FUNCTION_BLOCK OPCUA_CONNECT_13434D741E95123C0 (* Generic Interface Function Block Type *)
  (* Standard: 61499-2 *)
  (* Version 0.0, 20/09/2020, Administrator, nxtControl GmbH, Template *)
  PACKAGE Main;
  (* Compiler Cpp nxtControl builtin 1.0 *)
  {SET_ATTRIBUTE(Runtime.FBType.ImplementingType, Standard.OPCUAClient#DYNGEN_OPCUA_CONNECT)}
  {SET_ATTRIBUTE(Configuration.GenericFBType.InterfaceParams, Standard.OPCUAClient#CNTX:=1)}
  {SET_ATTRIBUTE(Configuration.FBType.IsKind.OPCUA_CLIENT, )}
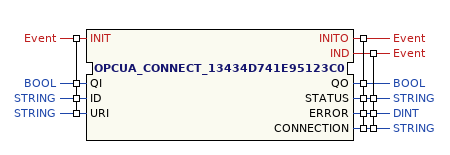
  EVENT_INPUT
    INIT WITH QI, ID, URI; (* Initialization or deinitialization of connection *)
  END_EVENT
  EVENT_OUTPUT
    INITO WITH QO, STATUS, ERROR, CONNECTION; (* Initialization or deinitialization confirmation event *)
    IND WITH STATUS, ERROR, CONNECTION; (* Indication of change in STATUS or ERROR or CONNECTION data outputs *)
  END_EVENT
  VAR_INPUT
    QI : BOOL; (* Input event qualifier *)
    ID : STRING; (* Connection ID; this ID should be unique within a device *)
    URI : STRING; (* URI of OPC UA server to which the client connects *)
  END_VAR
  VAR_OUTPUT
    QO : BOOL; (* Output event qualifier *)
    STATUS : STRING; (* Displays current connection status to the OPC UA server *)
    ERROR : DINT; (* Displays error code of service action associated with last event *)
    CONNECTION : STRING; (* Connection  ID; same as the ID input if the connection is successful otherwise empty. *)
  END_VAR
  EC_STATES
    START;
  END_STATES
END_FUNCTION_BLOCK
